(* CoDeSys 2.3 export: ST_TEMPERATUREUNIT.EXP *)

(* Data type *)
TYPE ST_TemperatureUnit :
STRUCT
	id: E_TemperatureUnit;
	unit: STRING;
	symbol: STRING;
	f1: REAL;
	f2: REAL;
	offset: REAL;
	scale: REAL;
	inventor: STRING;
END_STRUCT
END_TYPE
